PROGRAM MAIN
VAR
	ILD1420_Sensor1	: ILD1420;	// instance of ILD1420 Distance Senor
	ILD1420_Sensor2 : ILD1420;	// instance of ILD1420 Distance Senor
	
	lrDistance1 	: LREAL;		// var for distance 1 (could also be GVL)
	lrDistance2 	: LREAL;		// var for distance 1 (could also be GVL)
END_VAR

SerialComms_EL6021_ILD1420();		

ILD1420_Sensor1(RxBuffer := GVL_SerialBuffers.RxBufferEL[0]);		// init sensor 1
ILD1420_Sensor2(RxBuffer := GVL_SerialBuffers.RxBufferEL[1]);		// init sensor 2


lrDistance1 := ILD1420_Sensor1.lrDistance;
lrDistance2 := ILD1420_Sensor2.lrDistance;

GVL_HMI.rDist1 := lrDistance1;

END_PROGRAM

(* stored: Version 1.1.0.1, ProductVersion 3.1.4024.11
   POU MAIN: Id {62e43a78-46c8-44c8-9f1f-e8406f48095f}, SpecialFunc None *)
